// TIA Portal V21 export
// export: Created 2026-05-11T00:00:00.0000000Z, ExportSetting None, DisplayName Totally Integrated Automation Portal, DisplayVersion V21, DisplayName STEP 7 Professional, DisplayVersion V21
FUNCTION_BLOCK "MCPVerify_FB_LAD_v3"   // FB59989, LAD
TITLE = MCPVerify_FB_LAD_v3
{ S7_Optimized_Access := 'TRUE' }
// TON 实例在 FB.Static（TON_TIME）；PBox/Not/Lt — 安全 PLC 可用
// stored: AutoNumber false, MemoryReserve 50, SetENOAutomatically false
   VAR_INPUT
      Trig : Bool;
      PulseBit : Bool;
      NegIn : Bool;
      CmpA : Int;
      CmpB : Int;
   END_VAR
   VAR_OUTPUT
      OutTonQ : Bool;
      OutPulse : Bool;
      OutNot : Bool;
      OutLt : Bool;
   END_VAR
   VAR
      tonInst { S7_SetPoint := 'True'} : TON_TIME;
   END_VAR
   VAR_TEMP
      PulseWork : Bool;
   END_VAR
   VAR_TEMP   // added for the SCL form of the ladder/FBD networks
      _w1 : Bool;
   END_VAR
BEGIN

REGION Network 1: N1
   // N1 TON Static
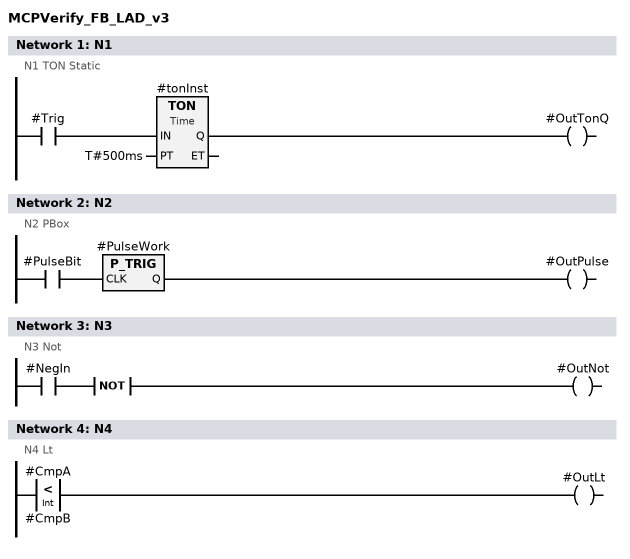
   RUNG wire#powerrail
      Contact( #Trig )
      { S7_Templates := "time_type := Time" } #tonInst.TON(pt := T#500ms, et =>)
      Coil( #OutTonQ )
   END_RUNG
   // the same network as SCL:
   #tonInst(IN := #Trig, PT := T#500ms);   // TON
   #OutTonQ := #tonInst.Q;
END_REGION

REGION Network 2: N2
   // N2 PBox
   RUNG wire#powerrail
      Contact( #PulseBit )
      P_Trig( #PulseWork )
      Coil( #OutPulse )
   END_RUNG
   // the same network as SCL:
   #_w1 := #PulseBit AND NOT #PulseWork;   // rising edge
   #PulseWork := #PulseBit;
   #OutPulse := #_w1;
END_REGION

REGION Network 3: N3
   // N3 Not
   RUNG wire#powerrail
      Contact( #NegIn )
      Not()
      Coil( #OutNot )
   END_RUNG
   // the same network as SCL:
   #OutNot := NOT #NegIn;
END_REGION

REGION Network 4: N4
   // N4 Lt
   RUNG wire#powerrail
      { S7_Templates := "SrcType := Int" } LT_Contact(in1 := #CmpA, in2 := #CmpB)
      Coil( #OutLt )
   END_RUNG
   // the same network as SCL:
   #OutLt := #CmpA < #CmpB;
END_REGION
END_FUNCTION_BLOCK
